PROGRAM PRG_ADSReadReq
VAR
	fbUA_Connect			: UA_Connect;
	SessionConnectInfo		: ST_UASessionConnectInfo;
	sOpcUA_URL				: STRING(MAX_STRING_LENGTH);
	nConnectionHdl			: DWORD;

	fbUA_GetNamespaceIndex 	: UA_GetNamespaceIndex;
	nNamespaceIndex			: UINT;
	
	fbUA_MethodCall_ADSReadReq	: UA_MethodCall_ADSReadReq;
	stADSReadRes				: ST_ADSReadRes;	// the Read variable is inside this struct
	
	stOutputArgInfo				: ARRAY [1..nNumberOfOutputArguments] OF ST_UAMethodArgInfo;
	
	fbUA_NodeReleaseHandle		: UA_NodeReleaseHandle;
	
	fbUA_Disconnect				: UA_Disconnect;
		
	bTest		: BOOL:= TRUE;
	bDone		: BOOL;
	bBusy		: BOOL;
	bError		: BOOL;
	nErrorID	: DWORD;
	iState		: INT;	
END_VAR
VAR CONSTANT
	nNumberOfOutputArguments	: UDINT := 1;
END_VAR


CASE iState OF
0:	(* idle *)
	IF bTest THEN
		bTest		:= FALSE;
		bError		:= FALSE;
		nErrorID	:= 0;

		(* Parameterize *)
		sOpcUA_URL						:= 'opc.tcp://localhost:4840';	(* OpcUA Url of the device with ip address *)

		SessionConnectInfo.tConnectTimeout 	:= t#1s;
		SessionConnectInfo.tSessionTimeout 	:= t#1s;
		SessionConnectInfo.sApplicationName	:= '';
//		SessionConnectInfo.sApplicationUri 	:= '';
		SessionConnectInfo.eSecurityMode 		:= eUASecurityMsgMode_None;
		SessionConnectInfo.eSecurityPolicyUri 	:= eUASecurityPolicy_None;
		SessionConnectInfo.eTransportProfileUri := eUATransportProfileUri_UATcp;

		iState	:= iState + 1;	(* open ua session *)
	END_IF

1:	(* open UA session *)
	fbUA_Connect(
		Execute				:= TRUE,
		ServerURL			:= sOpcUA_URL,
		SessionConnectInfo	:= SessionConnectInfo,
		Timeout				:= T#5S,
		ConnectionHdl		=> nConnectionHdl
	);

	IF NOT fbUA_Connect.Busy THEN
		fbUA_Connect(Execute := FALSE);

		IF NOT fbUA_Connect.Error THEN
			(* session open *)
			iState := iState + 1;	(* get namespace index *)
		ELSE
			bError			:= TRUE;
			nErrorID		:= fbUA_Connect.ErrorID;
			nConnectionHdl	:= 0;
			iState 			:= 0; (* idle *)
		END_IF
	END_IF


2:	(* GetNS Index *)
	fbUA_GetNamespaceIndex(
		Execute			:= TRUE,
		ConnectionHdl	:= nConnectionHdl,
		NamespaceUri	:= 'ADSAMS',
		NamespaceIndex	=> nNamespaceIndex
	);

	IF NOT fbUA_GetNamespaceIndex.Busy THEN
		fbUA_GetNamespaceIndex(Execute := FALSE);

		IF NOT fbUA_GetNamespaceIndex.Error THEN
			(* session closed *)
			iState 		:= iState + 1; (* method *)
		ELSE
			bError		:= TRUE;
			nErrorID	:= fbUA_GetNamespaceIndex.ErrorID;
			iState 		:= 4; (* close session *)
		END_IF
	END_IF

3:	(*  Method  *)
	stOutputArgInfo[1].nLenData := SIZEOF(stADSReadRes.nReadData); 
	fbUA_MethodCall_ADSReadReq(
		bExecute		:= TRUE,
		nConnectionHdl	:= nConnectionHdl,
		nNamespaceIndex	:= nNamespaceIndex,
		sNetID			:= '127.0.0.1.1.1',
		nPort			:= 851,
		nIndexGroup		:= 16#4020,
		nIndexOffset	:= 0,
		pOutputArgInfoAndData 	:= ADR(stADSReadRes),		// buffer for output argument info and output data
		cbOutputArgInfoAndData	:= SIZEOF(stADSReadRes),	// size output argument info + Data
		cbReadData		:= SIZEOF(stADSReadRes.nReadData),	//size of Data only
		nNumberOfOutputArguments:= nNumberOfOutputArguments,
		pOutputArgInfo	:= ADR(stOutputArgInfo),
		cbOutputArgInfo	:= SIZEOF(stOutputArgInfo)		
		);


	IF NOT fbUA_MethodCall_ADSReadReq.bBusy THEN
		fbUA_MethodCall_ADSReadReq(bExecute := FALSE);
		IF NOT fbUA_MethodCall_ADSReadReq.bError THEN
			(* session closed *)
			iState 		:= iState + 1; (* close session *)
		ELSE
			bError		:= TRUE;
			nErrorID	:= fbUA_MethodCall_ADSReadReq.nErrorID;
			iState 		:= 4; (* close session *)
		END_IF
	END_IF


4:	(* close session *)
	fbUA_Disconnect(
		Execute			:= TRUE,
		ConnectionHdl	:= nConnectionHdl
	);

	IF NOT fbUA_Disconnect.Busy THEN
		fbUA_Disconnect(Execute := FALSE);
		bBusy := FALSE;
		IF NOT fbUA_Disconnect.Error THEN
			(* session closed *)
			iState 		:= 0; (* idle *)
			IF NOT bError THEN 
				bDone 	:= TRUE;
			END_IF
		ELSE
			bError			:= TRUE;
			nErrorID		:= fbUA_Disconnect.ErrorID;
			iState 			:= 0; (* idle *)
			nConnectionHdl	:= 0;
		END_IF
	END_IF
END_CASE

END_PROGRAM

(* stored: Version 1.1.0.1, ProductVersion 3.1.4022.6
   POU PRG_ADSReadReq: Id {c9607e7a-4215-4f37-91f4-6d3efb6321f8}, SpecialFunc None *)
